FUNCTION_BLOCK T_Stop IMPLEMENTS I_Stop
VAR
	axRef : REFERENCE TO AXIS_REF;
	_stop : MC_Stop;
END_VAR

IF NOT __ISVALIDREF( axRef ) THEN
	RETURN;
END_IF

_stop( Axis := axRef );
_stop.Execute R= 
	_stop.Done 
	OR axRef.Status.Disabled;

PROPERTY PUBLIC Busy : BOOL
GET
END_GET
END_PROPERTY

PROPERTY PUBLIC Error : BOOL
GET
Error := 
	_stop.Error 
	OR NOT __ISVALIDREF( axRef );
END_GET
END_PROPERTY

METHOD PUBLIC Parameterise : BOOL
VAR_INPUT
	deceleration : LREAL;
	jerk : LREAL;
END_VAR
IF Busy THEN
	RETURN;
END_IF

_stop.Deceleration := deceleration;
_stop.Jerk := jerk;
Parameterise := TRUE;
END_METHOD

METHOD PUBLIC RegisterAxis : BOOL
VAR_IN_OUT
	axisRef : AXIS_REF;
END_VAR
IF Busy THEN // Error
	RETURN;
END_IF

axRef REF= axisRef;
END_METHOD

METHOD Stop
_stop.Execute := TRUE;
END_METHOD

END_FUNCTION_BLOCK

(* stored: Version 1.1.0.1, ProductVersion 3.1.4024.3
   POU T_Stop: Id {58c15be9-02d8-461a-b27e-2c5b2802f508}, SpecialFunc None
   Property Busy: Id {a7eb2eea-d5a4-40de-b4a0-87d9bfb35875}
   Get Get: Id {2ccecaef-c25a-4a37-ac73-bdeed39cf0c7}
   Property Error: Id {796f8ada-5229-4bbd-bb3b-2927305af202}
   Get Get: Id {da6b8ff1-932a-4abd-8341-6b76d0d020ca}
   Method Parameterise: Id {b3267be7-b734-4dac-96c1-edd142025da5}
   Method RegisterAxis: Id {61d05de7-464e-4679-aef4-91ac961d27b8}
   Method Stop: Id {6c737fe9-781b-4ebb-9972-ba15d8a8c3cc} *)
